FUNCTION_BLOCK EL5101
VAR
	_io : EL5101_Data;
	{attribute addProperty Name "WcState"}
	_wcState : WcStateInputToggle;
	{attribute addProperty Name "Info data"}
	_infoData : InfoDataAdsDC;
END_VAR

PROPERTY IO : REFERENCE TO EL5101_Data
GET
IO REF= _io;
END_GET
END_PROPERTY

PROPERTY WcState : REFERENCE TO WcStateInputToggle
GET
WcState REF= _wcState;
END_GET
END_PROPERTY

END_FUNCTION_BLOCK

(* stored: Version 1.1.0.1, ProductVersion 3.1.4024.9
   POU EL5101: Id {8491a08c-e246-0e92-32c9-75a9c424591a}, SpecialFunc None
   Property IO: Id {70634c02-1c5a-00f1-394f-8fe5fecb7888}
   Get Get: Id {2e2297fa-10a3-0f28-2b8f-44e87405ca21}
   Property WcState: Id {08fd0c56-30cc-07a2-058c-b5f9c493ea0b}
   Get Get: Id {7c1e9618-ecec-0fdb-309a-f2b6dc5281ce} *)
